PROGRAM P_Dimmers_RB2
VAR
	fbDALIV2Dimmer2Switch_RB2_1		: FB_DALIV2Dimmer2Switch;
	nActualLEvelMasterDev_1			: BYTE;
	bBusy_1							: BOOL;
	bError_1						: BOOL;
	nErrorId_1						: UDINT;
	
	
	fbDALIV2Dimmer2Switch_RB2_2		: FB_DALIV2Dimmer2Switch;
	nActualLEvelMasterDev_2			: BYTE;
	bBusy_2							: BOOL;
	bError_2						: BOOL;
	nErrorId_2						: UDINT;
	
	
	fbDALIV2Dimmer2Switch_RB2_3		: FB_DALIV2Dimmer2Switch;
	nActualLEvelMasterDev_3			: BYTE;
	bBusy_3							: BOOL;
	bError_3						: BOOL;
	nErrorId_3						: UDINT;
	
	fbDALIV2Dimmer2Switch_RB2_4		: FB_DALIV2Dimmer2Switch;
	nActualLEvelMasterDev_4			: BYTE;
	bBusy_4							: BOOL;
	bError_4						: BOOL;
	nErrorId_4						: UDINT;
	
	fbDALIV2Dimmer2Switch_RB2_5		: FB_DALIV2Dimmer2Switch;
	nActualLEvelMasterDev_5			: BYTE;
	bBusy_5							: BOOL;
	bError_5						: BOOL;
	nErrorId_5						: UDINT;
	
	fbDALIV2Dimmer2Switch_RB2_6		: FB_DALIV2Dimmer2Switch;
	nActualLEvelMasterDev_6			: BYTE;
	bBusy_6							: BOOL;
	bError_6						: BOOL;
	nErrorId_6						: UDINT;
	
	fbDALIV2Dimmer2Switch_RB2_7		: FB_DALIV2Dimmer2Switch;
	nActualLEvelMasterDev_7			: BYTE;
	bBusy_7							: BOOL;
	bError_7						: BOOL;
	nErrorId_7						: UDINT;
	
	fbDALIV2Dimmer2Switch_RB2_8		: FB_DALIV2Dimmer2Switch;
	nActualLEvelMasterDev_8			: BYTE;
	bBusy_8							: BOOL;
	bError_8						: BOOL;
	nErrorId_8						: UDINT;
	
END_VAR

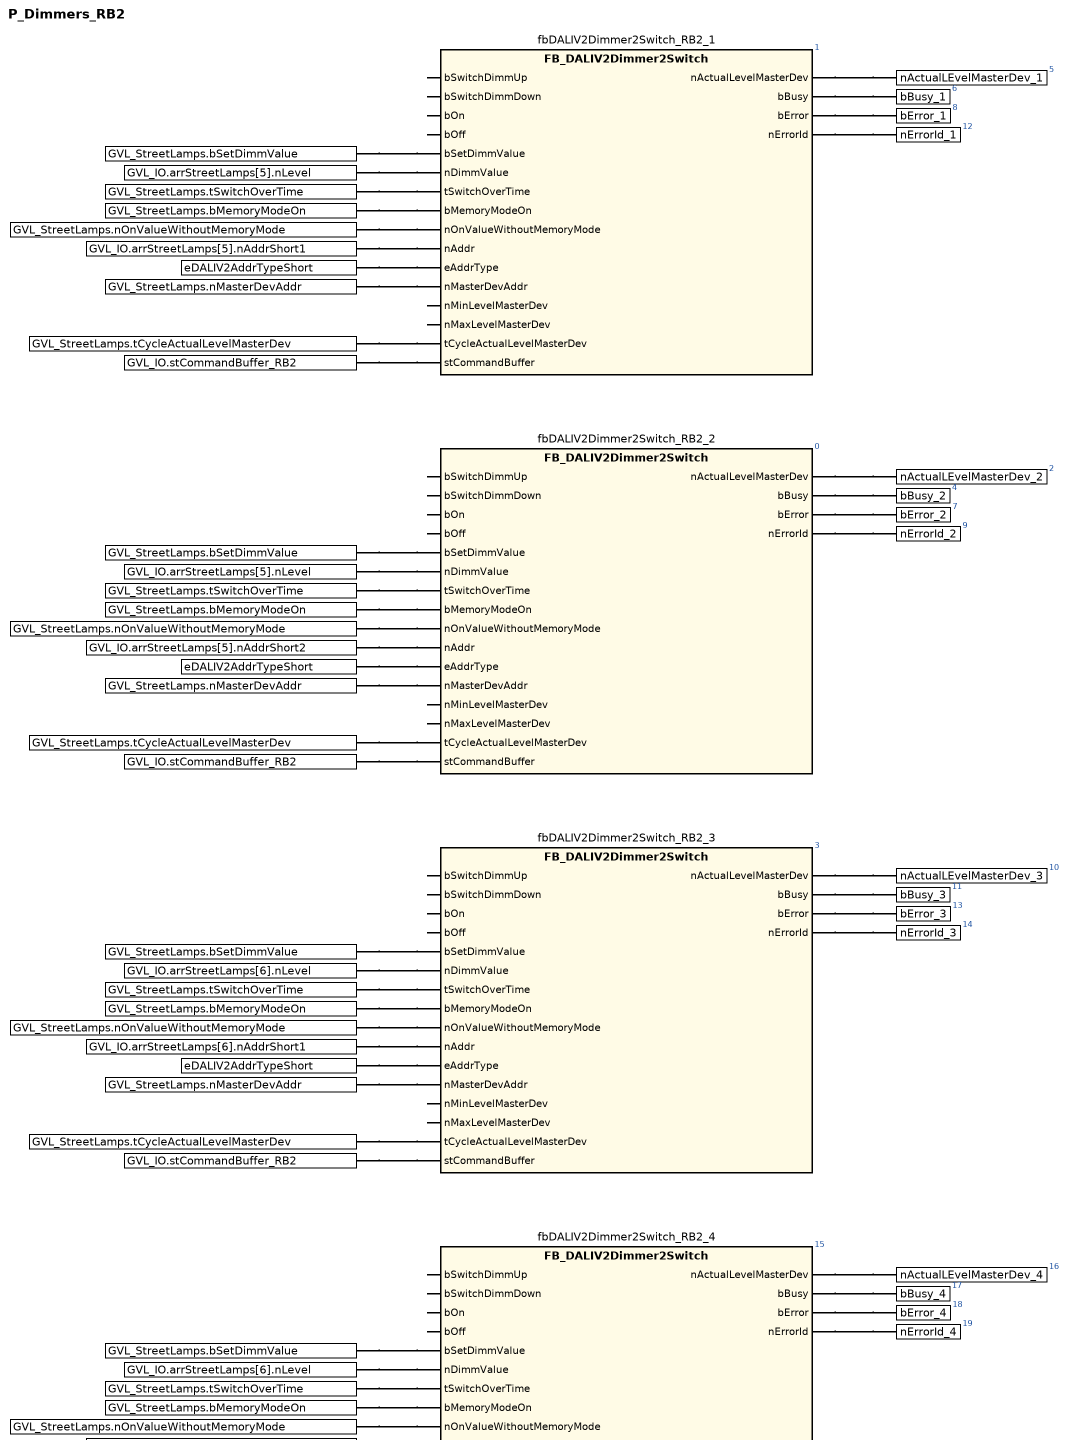
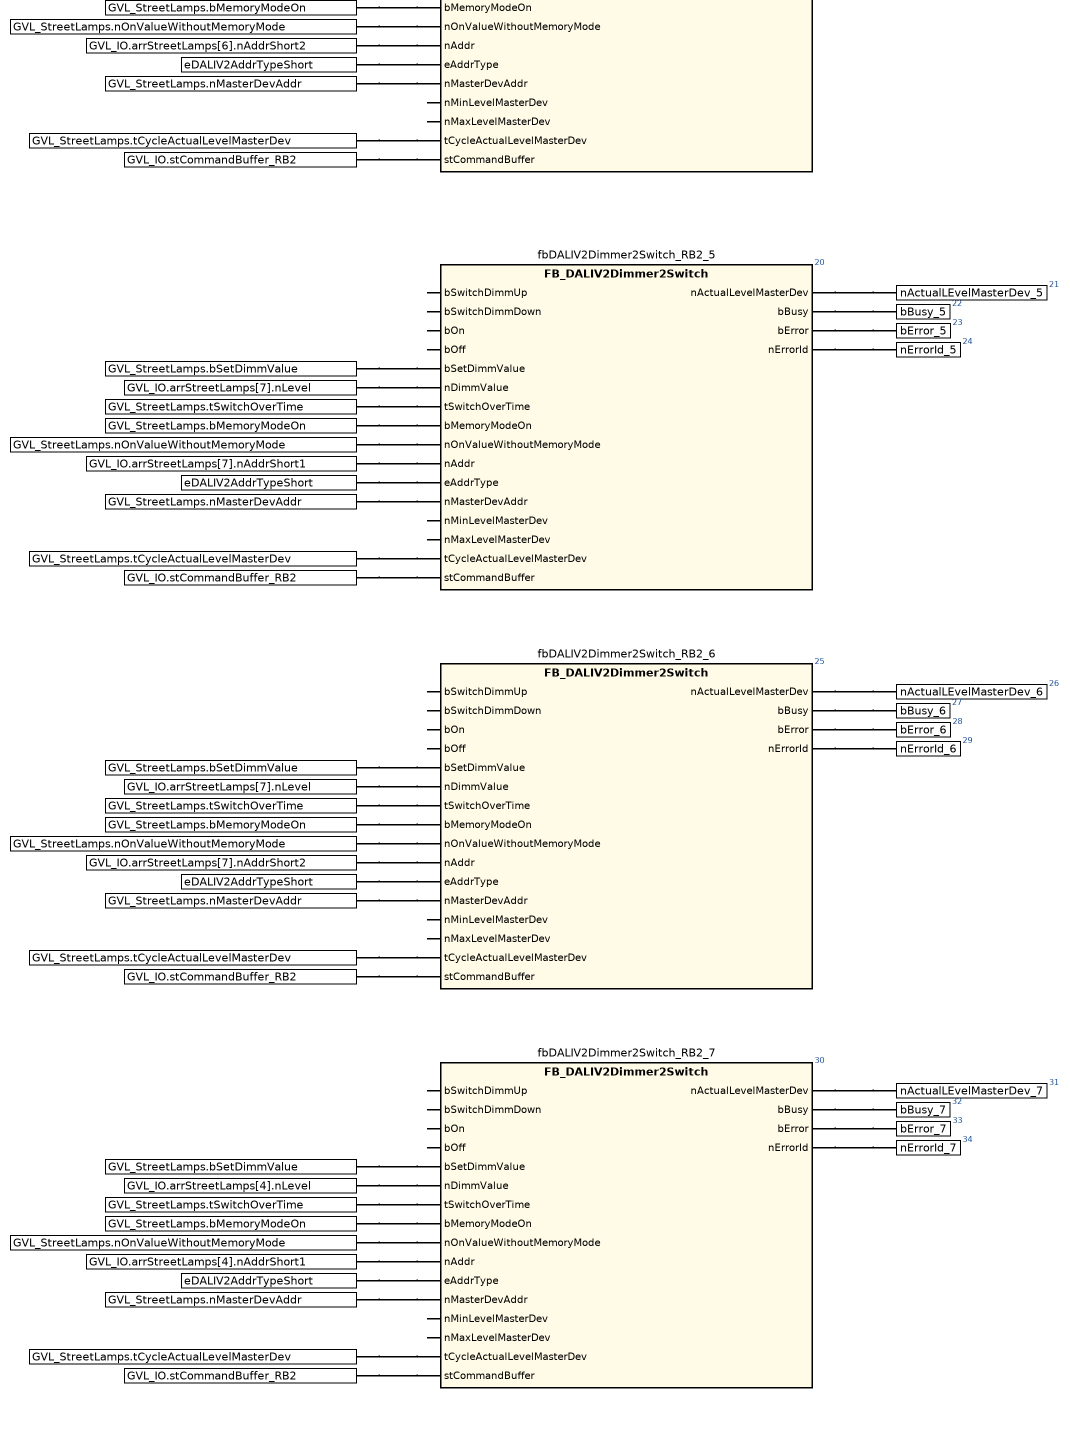
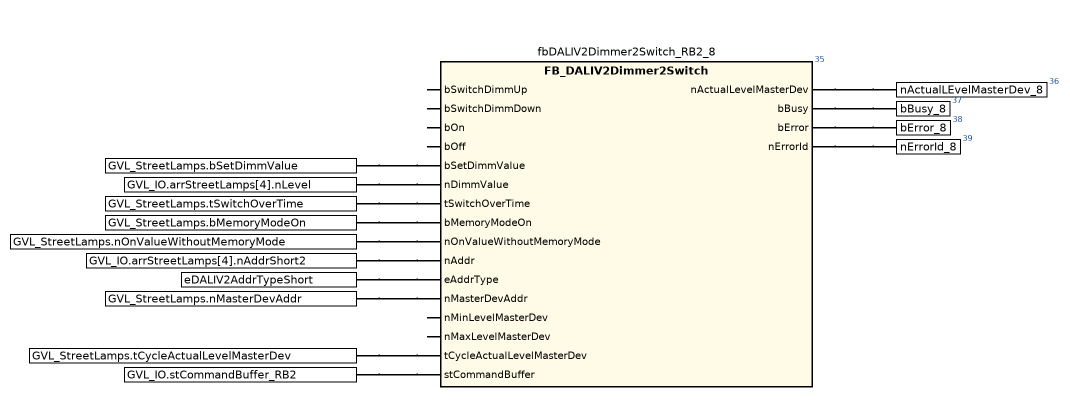
fbDALIV2Dimmer2Switch_RB2_2(
    bSetDimmValue := GVL_StreetLamps.bSetDimmValue,
    nDimmValue := GVL_IO.arrStreetLamps[5].nLevel,
    tSwitchOverTime := GVL_StreetLamps.tSwitchOverTime,
    bMemoryModeOn := GVL_StreetLamps.bMemoryModeOn,
    nOnValueWithoutMemoryMode := GVL_StreetLamps.nOnValueWithoutMemoryMode,
    nAddr := GVL_IO.arrStreetLamps[5].nAddrShort2,
    eAddrType := eDALIV2AddrTypeShort,
    nMasterDevAddr := GVL_StreetLamps.nMasterDevAddr,
    tCycleActualLevelMasterDev := GVL_StreetLamps.tCycleActualLevelMasterDev,
    stCommandBuffer := GVL_IO.stCommandBuffer_RB2); // FB_DALIV2Dimmer2Switch
fbDALIV2Dimmer2Switch_RB2_1(
    bSetDimmValue := GVL_StreetLamps.bSetDimmValue,
    nDimmValue := GVL_IO.arrStreetLamps[5].nLevel,
    tSwitchOverTime := GVL_StreetLamps.tSwitchOverTime,
    bMemoryModeOn := GVL_StreetLamps.bMemoryModeOn,
    nOnValueWithoutMemoryMode := GVL_StreetLamps.nOnValueWithoutMemoryMode,
    nAddr := GVL_IO.arrStreetLamps[5].nAddrShort1,
    eAddrType := eDALIV2AddrTypeShort,
    nMasterDevAddr := GVL_StreetLamps.nMasterDevAddr,
    tCycleActualLevelMasterDev := GVL_StreetLamps.tCycleActualLevelMasterDev,
    stCommandBuffer := GVL_IO.stCommandBuffer_RB2); // FB_DALIV2Dimmer2Switch
nActualLEvelMasterDev_2 := fbDALIV2Dimmer2Switch_RB2_2.nActualLevelMasterDev;
fbDALIV2Dimmer2Switch_RB2_3(
    bSetDimmValue := GVL_StreetLamps.bSetDimmValue,
    nDimmValue := GVL_IO.arrStreetLamps[6].nLevel,
    tSwitchOverTime := GVL_StreetLamps.tSwitchOverTime,
    bMemoryModeOn := GVL_StreetLamps.bMemoryModeOn,
    nOnValueWithoutMemoryMode := GVL_StreetLamps.nOnValueWithoutMemoryMode,
    nAddr := GVL_IO.arrStreetLamps[6].nAddrShort1,
    eAddrType := eDALIV2AddrTypeShort,
    nMasterDevAddr := GVL_StreetLamps.nMasterDevAddr,
    tCycleActualLevelMasterDev := GVL_StreetLamps.tCycleActualLevelMasterDev,
    stCommandBuffer := GVL_IO.stCommandBuffer_RB2); // FB_DALIV2Dimmer2Switch
bBusy_2 := fbDALIV2Dimmer2Switch_RB2_2.bBusy;
nActualLEvelMasterDev_1 := fbDALIV2Dimmer2Switch_RB2_1.nActualLevelMasterDev;
bBusy_1 := fbDALIV2Dimmer2Switch_RB2_1.bBusy;
bError_2 := fbDALIV2Dimmer2Switch_RB2_2.bError;
bError_1 := fbDALIV2Dimmer2Switch_RB2_1.bError;
nErrorId_2 := fbDALIV2Dimmer2Switch_RB2_2.nErrorId;
nActualLEvelMasterDev_3 := fbDALIV2Dimmer2Switch_RB2_3.nActualLevelMasterDev;
bBusy_3 := fbDALIV2Dimmer2Switch_RB2_3.bBusy;
nErrorId_1 := fbDALIV2Dimmer2Switch_RB2_1.nErrorId;
bError_3 := fbDALIV2Dimmer2Switch_RB2_3.bError;
nErrorId_3 := fbDALIV2Dimmer2Switch_RB2_3.nErrorId;
fbDALIV2Dimmer2Switch_RB2_4(
    bSetDimmValue := GVL_StreetLamps.bSetDimmValue,
    nDimmValue := GVL_IO.arrStreetLamps[6].nLevel,
    tSwitchOverTime := GVL_StreetLamps.tSwitchOverTime,
    bMemoryModeOn := GVL_StreetLamps.bMemoryModeOn,
    nOnValueWithoutMemoryMode := GVL_StreetLamps.nOnValueWithoutMemoryMode,
    nAddr := GVL_IO.arrStreetLamps[6].nAddrShort2,
    eAddrType := eDALIV2AddrTypeShort,
    nMasterDevAddr := GVL_StreetLamps.nMasterDevAddr,
    tCycleActualLevelMasterDev := GVL_StreetLamps.tCycleActualLevelMasterDev,
    stCommandBuffer := GVL_IO.stCommandBuffer_RB2); // FB_DALIV2Dimmer2Switch
nActualLEvelMasterDev_4 := fbDALIV2Dimmer2Switch_RB2_4.nActualLevelMasterDev;
bBusy_4 := fbDALIV2Dimmer2Switch_RB2_4.bBusy;
bError_4 := fbDALIV2Dimmer2Switch_RB2_4.bError;
nErrorId_4 := fbDALIV2Dimmer2Switch_RB2_4.nErrorId;
fbDALIV2Dimmer2Switch_RB2_5(
    bSetDimmValue := GVL_StreetLamps.bSetDimmValue,
    nDimmValue := GVL_IO.arrStreetLamps[7].nLevel,
    tSwitchOverTime := GVL_StreetLamps.tSwitchOverTime,
    bMemoryModeOn := GVL_StreetLamps.bMemoryModeOn,
    nOnValueWithoutMemoryMode := GVL_StreetLamps.nOnValueWithoutMemoryMode,
    nAddr := GVL_IO.arrStreetLamps[7].nAddrShort1,
    eAddrType := eDALIV2AddrTypeShort,
    nMasterDevAddr := GVL_StreetLamps.nMasterDevAddr,
    tCycleActualLevelMasterDev := GVL_StreetLamps.tCycleActualLevelMasterDev,
    stCommandBuffer := GVL_IO.stCommandBuffer_RB2); // FB_DALIV2Dimmer2Switch
nActualLEvelMasterDev_5 := fbDALIV2Dimmer2Switch_RB2_5.nActualLevelMasterDev;
bBusy_5 := fbDALIV2Dimmer2Switch_RB2_5.bBusy;
bError_5 := fbDALIV2Dimmer2Switch_RB2_5.bError;
nErrorId_5 := fbDALIV2Dimmer2Switch_RB2_5.nErrorId;
fbDALIV2Dimmer2Switch_RB2_6(
    bSetDimmValue := GVL_StreetLamps.bSetDimmValue,
    nDimmValue := GVL_IO.arrStreetLamps[7].nLevel,
    tSwitchOverTime := GVL_StreetLamps.tSwitchOverTime,
    bMemoryModeOn := GVL_StreetLamps.bMemoryModeOn,
    nOnValueWithoutMemoryMode := GVL_StreetLamps.nOnValueWithoutMemoryMode,
    nAddr := GVL_IO.arrStreetLamps[7].nAddrShort2,
    eAddrType := eDALIV2AddrTypeShort,
    nMasterDevAddr := GVL_StreetLamps.nMasterDevAddr,
    tCycleActualLevelMasterDev := GVL_StreetLamps.tCycleActualLevelMasterDev,
    stCommandBuffer := GVL_IO.stCommandBuffer_RB2); // FB_DALIV2Dimmer2Switch
nActualLEvelMasterDev_6 := fbDALIV2Dimmer2Switch_RB2_6.nActualLevelMasterDev;
bBusy_6 := fbDALIV2Dimmer2Switch_RB2_6.bBusy;
bError_6 := fbDALIV2Dimmer2Switch_RB2_6.bError;
nErrorId_6 := fbDALIV2Dimmer2Switch_RB2_6.nErrorId;
fbDALIV2Dimmer2Switch_RB2_7(
    bSetDimmValue := GVL_StreetLamps.bSetDimmValue,
    nDimmValue := GVL_IO.arrStreetLamps[4].nLevel,
    tSwitchOverTime := GVL_StreetLamps.tSwitchOverTime,
    bMemoryModeOn := GVL_StreetLamps.bMemoryModeOn,
    nOnValueWithoutMemoryMode := GVL_StreetLamps.nOnValueWithoutMemoryMode,
    nAddr := GVL_IO.arrStreetLamps[4].nAddrShort1,
    eAddrType := eDALIV2AddrTypeShort,
    nMasterDevAddr := GVL_StreetLamps.nMasterDevAddr,
    tCycleActualLevelMasterDev := GVL_StreetLamps.tCycleActualLevelMasterDev,
    stCommandBuffer := GVL_IO.stCommandBuffer_RB2); // FB_DALIV2Dimmer2Switch
nActualLEvelMasterDev_7 := fbDALIV2Dimmer2Switch_RB2_7.nActualLevelMasterDev;
bBusy_7 := fbDALIV2Dimmer2Switch_RB2_7.bBusy;
bError_7 := fbDALIV2Dimmer2Switch_RB2_7.bError;
nErrorId_7 := fbDALIV2Dimmer2Switch_RB2_7.nErrorId;
fbDALIV2Dimmer2Switch_RB2_8(
    bSetDimmValue := GVL_StreetLamps.bSetDimmValue,
    nDimmValue := GVL_IO.arrStreetLamps[4].nLevel,
    tSwitchOverTime := GVL_StreetLamps.tSwitchOverTime,
    bMemoryModeOn := GVL_StreetLamps.bMemoryModeOn,
    nOnValueWithoutMemoryMode := GVL_StreetLamps.nOnValueWithoutMemoryMode,
    nAddr := GVL_IO.arrStreetLamps[4].nAddrShort2,
    eAddrType := eDALIV2AddrTypeShort,
    nMasterDevAddr := GVL_StreetLamps.nMasterDevAddr,
    tCycleActualLevelMasterDev := GVL_StreetLamps.tCycleActualLevelMasterDev,
    stCommandBuffer := GVL_IO.stCommandBuffer_RB2); // FB_DALIV2Dimmer2Switch
nActualLEvelMasterDev_8 := fbDALIV2Dimmer2Switch_RB2_8.nActualLevelMasterDev;
bBusy_8 := fbDALIV2Dimmer2Switch_RB2_8.bBusy;
bError_8 := fbDALIV2Dimmer2Switch_RB2_8.bError;
nErrorId_8 := fbDALIV2Dimmer2Switch_RB2_8.nErrorId;

END_PROGRAM

(* stored: Version 1.1.0.1, ProductVersion 3.1.4024.5
   POU P_Dimmers_RB2: Id {661592a3-149f-4a76-8033-62ad87a0efc8}, SpecialFunc None *)
